FUNCTION_BLOCK Test_TStreamAdd_Read_BLOB EXTENDS TUnitTestBase
VAR
    Stream : TStream(StreamLength := 2);
    Now : TIMESTRUCT := (wDay := 23, wMonth := 12, wYear := 1945, wHour := 22, wMinute := 20, wSecond := 18);
    NowFromStream : TIMESTRUCT;
    
    LREAL_Value : LREAL := 1.234;
END_VAR



Stream.Init(2);

Stream.Add_BLOB(Now);
Stream.Add_LREAL(LREAL_Value);
    
Stream.Seek(0);

Stream.Read_BLOB(NowFromStream);

Assertion.AssertEquals_BLOB(
    Expected := Now,
    Actual := NowFromStream,
    VariableName := 'NowFromStream');
    
Assertion.AssertEquals_LREAL(
    Expected := 1.234,
    Actual := Stream.Read_LREAL(),
    Delta  := 0.000001,
    VariableName := 'Stream.Read_LREAL()');
    
    
TestFinished();

END_FUNCTION_BLOCK

(* stored: Version 1.1.0.1, ProductVersion 3.1.4024.4
   POU Test_TStreamAdd_Read_BLOB: Id {857ecb43-3569-4de4-8aef-bebb116450cf}, SpecialFunc None *)
